TYPE ST_HMI_PrinterStatus :
STRUCT
	sPrinterName					: STRING(30);
(* read only *)
	bPrinterReady					: BOOL;
	bActivePrinter					: BOOL;
	bPrinterInService				: BOOL;		(*printer Avalable*)
	bPrinterSelected				: BOOL;
	bDataReady					: BOOL;
	bHomePosition				: BOOL;
	bLabelPrinted					: BOOL;
	bReadyToApply				: BOOL;
	bApplyDone					: BOOL;
	bSummaryWarning				: BOOL;
	bPrinterError					: BOOL;

	Q								: ST_PRINTER_OUT;

END_STRUCT
END_TYPE

(* stored: Version 1.1.0.1, ProductVersion 3.1.4024.15
   DUT ST_HMI_PrinterStatus: Id {9d0a28d8-bdec-4b81-afcd-dc3b50bf8822} *)
